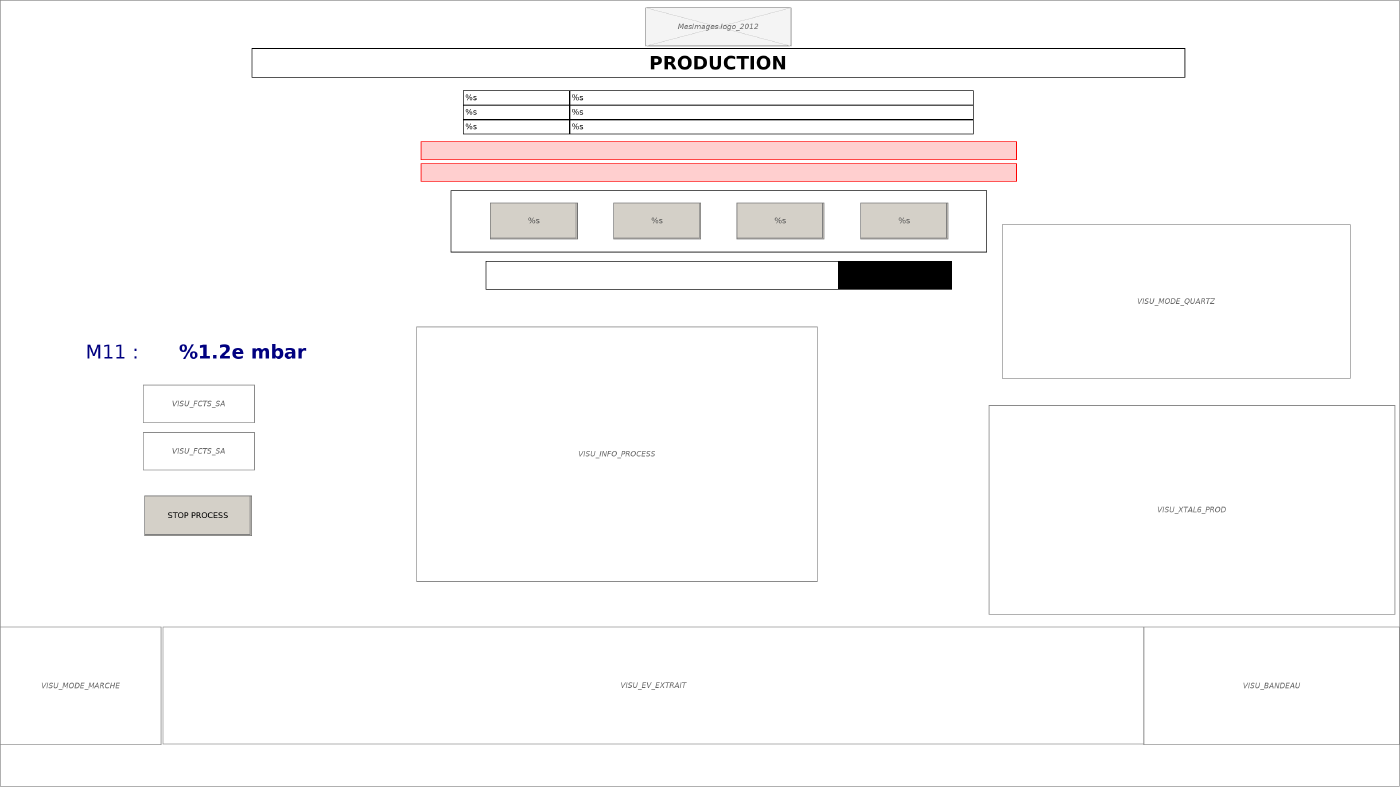
VISUALIZATION SYN_EXEC_PROC  // 1920x1080, background image fond_blanc_1280_1024
    Frame (223,860 1346x161)
        shows VISU_EV_EXTRAIT()
    Frame (1568,860 352x162)
        shows VISU_BANDEAU(m_Input_MACHINE := Global_Variables.MACHINE)
    Frame (0,860 221x162)
        shows VISU_MODE_MARCHE(m_Input_MACHINE := .MACHINE)
    RoundedRectangle (345,66 1280x40), "PRODUCTION"
    Group (635,124 700x60)
        Rectangle (0,0 146x20), "%s", text list: 'TextList_Process', text index: 0
        Rectangle (0,20 146x20), "%s", text list: 'TextList_Process', text index: 1
        Rectangle (0,40 146x20), "%s", text list: 'TextList_Process', text index: 2
        Rectangle (146,0 554x20), "%s", text variable: EXECPROC.PRM_PROCESS_NAME, text index: 0
        Rectangle (146,20 554x20), "%s", text variable: EXECPROC.STATE_STEP_TEXT, text index: 0
        Rectangle (146,40 554x20), "%s", text variable: MAIN.STEP_EMPILEMENT.STATE_LAYER_TEXT, text index: 0
    Group (618,261 735x85)
        RoundedRectangle (0,0 735x85)
        Button (54,17 120x50), "%s", input disabled if: (NOT MACHINE.AUTOR_Start_Prod_Ihm OR PRG_SEC.VERROU OR NOT PRG_User.ACTU_USER.PRODUCTION) OR MACHINE.STATE_Prod, text list: 'TextList_Process', text index: 3
            tap MAIN.bStartVerif
        Button (223,17 120x50), "%s", input disabled if: NOT (PRG_USER.ACTU_USER.PRODUCTION AND MACHINE.AUTOR_Stop_Prod_Ihm), text list: 'TextList_Process', text index: 4
            toggle MACHINE.M_Stop_Prod
        Button (392,17 120x50), "%s", input disabled if: NOT (PRG_USER.ACTU_USER.PRODUCTION AND MACHINE.AUTOR_Inter_Prod_ihm), text list: 'TextList_Process', text index: 5
            toggle MACHINE.M_inter_Prod
        Button (562,17 120x50), "%s", input disabled if: NOT (PRG_USER.ACTU_USER.PRODUCTION AND MACHINE.AUTOR_Repris_Prod_ihm), text list: 'TextList_Process', text index: 6
            toggle MACHINE.M_Reprise_Prod
    Frame (571,448 550x350), invisible if: NOT Global_Variables.MACHINE.STATE_Prod
        shows VISU_INFO_PROCESS()
    Image (885,10 200x53), image: MesImages.logo_2012
    Frame (196,528 153x52)
        shows VISU_FCTS_SA(m_Input_ID_XML := 4, m_Input_UserRight := PRG_USER.ACTU_USER.PRODUCTION AND NOT MACHINE.STATE_Prod AND NOT INIT_MACHINE.OP_INIT.EC, m_Input_Operation := PRG_POMPAGE.POMPAGE.OP_Ventilation)
    Frame (196,593 153x52)
        shows VISU_FCTS_SA(m_Input_ID_XML := 0, m_Input_UserRight := PRG_USER.ACTU_USER.PRODUCTION AND NOT MACHINE.STATE_Prod AND NOT INIT_MACHINE.OP_INIT.EC, m_Input_Operation := PRG_POMPAGE.POMPAGE.OP_Pompage_Sec)
    Button (198,680 147x55), "STOP PROCESS", invisible if: PRG_USER.ACTU_USER.MAINTENANCE OR NOT INIT_MACHINE.STATE_ABORT
        tap INIT_MACHINE.M_Stop_Procedure
    Group (666,358 639x39)
        Rectangle (0,0 484x39), text list: 'TextList_EcoMode', text index: 12
        Rectangle (484,0 155x39), colour toggle: MACHINE.PRM_EXEC_PROC_WEEKEND, input disabled if: NOT Global_Variables.PRG_USER.ACTU_USER.PRODUCTION
            toggle MACHINE.PRM_EXEC_PROC_WEEKEND
    Frame (1374,308 478x211)
        shows VISU_MODE_QUARTZ(m_input_Mode_Quartz := MODE_QUARTZ_PROD)
    Frame (1356,556 557x287)
        shows VISU_XTAL6_PROD(m_Input_XTAL6 := PRG_EVAP.QZ1)
    Rectangle (114,463 80x40), "M11 :"
    Rectangle (208,463 250x40), "%1.2e mbar", text variable: Global_Variables.PRG_POMPAGE.M11.STATE_Pression
    Group (577,194 817x55)
        Rectangle (0,0 817x25), invisible if: NOT MACHINE.DEF_Presence_TrAC.DEF, text list: 'TextList_Basiques', text index: 20
        Rectangle (0,30 817x25), invisible if: NOT MACHINE.DEF_Presence_ACSoft.DEF, text list: 'TextList_Basiques', text index: 21
END_VISUALIZATION

(* stored: Version 1.1.0.1, ProductVersion 3.1.4024.12
   Visu SYN_EXEC_PROC: Id {cef2b832-7432-4648-8ec8-10f9d7146113} *)
